% RSLogix 500 project TANK_ANAL_BAK001.RSS, saved by version 8.30.00.16 %
PROJECT "UNTITLED"    % processor: Bul.1763 MicroLogix 1100 Series B %

PROGRAM FILES
  LAD 2 "MAIN"  3 rungs
  LAD 3 "ANALOG IO"  4 rungs
  LAD 4 "CONTROLS"  5 rungs

DATA FILES
  O0 OUTPUT  5 elements
  I1 INPUT  14 elements
  S2 STATUS  66 elements
  B3 BINARY  1 elements
  T4 TIMER  2 elements
  C5 COUNTER  1 elements
  R6 CONTROL  1 elements
  N7 INTEGER  1 elements
  F8 FLOAT  1 elements

LADDER 2 "MAIN"
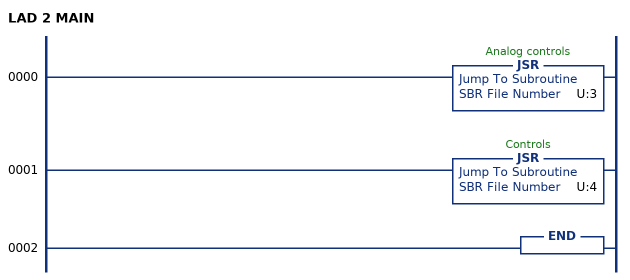
% Rung: 0 %
SOR JSR U:3 EOR
%   U:3  "Analog controls" %
% Rung: 1 %
SOR JSR U:4 EOR
%   U:4  "Controls" %
% Rung: 2 %
SOR END EOR

LADDER 3 "ANALOG IO"
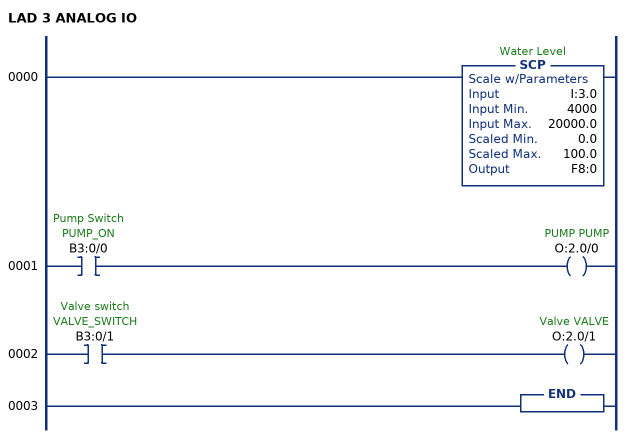
% Rung: 0 %
SOR SCP I:3.0 4000 20000.0 0.0 100.0 F8:0 EOR
%   I:3.0  WATER_LEVEL  "Water Level" %
%   F8:0  "Water Level" %
% Rung: 1 %
SOR XIC B3:0/0 OTE O:2.0/0 EOR
%   B3:0/0  PUMP_ON  "Pump Switch" %
%   O:2.0/0  PUMP  "PUMP" %
% Rung: 2 %
SOR XIC B3:0/1 OTE O:2.0/1 EOR
%   B3:0/1  VALVE_SWITCH  "Valve switch" %
%   O:2.0/1  VALVE  "Valve" %
% Rung: 3 %
SOR END EOR

LADDER 4 "CONTROLS"
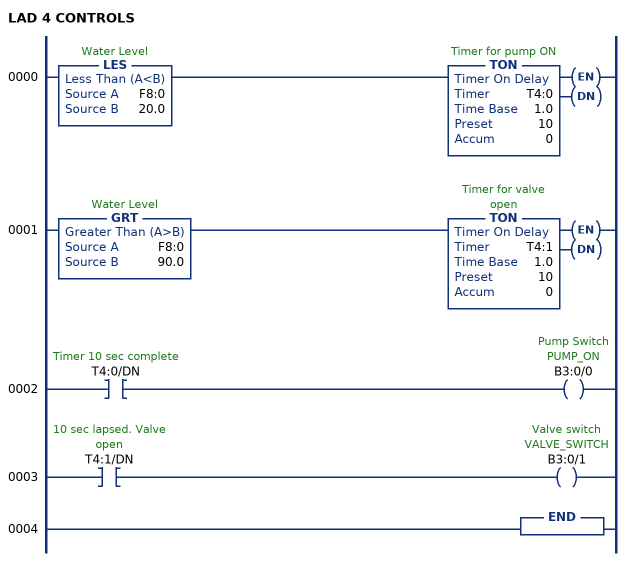
% Rung: 0 %
SOR LES F8:0 20.0 TON T4:0 1.0 10 0 EOR
%   F8:0  "Water Level" %
%   T4:0  "Timer for pump ON" %
% Rung: 1 %
SOR GRT F8:0 90.0 TON T4:1 1.0 10 0 EOR
%   F8:0  "Water Level" %
%   T4:1  "Timer for valve open" %
% Rung: 2 %
SOR XIC T4:0/DN OTE B3:0/0 EOR
%   T4:0/DN  "Timer 10 sec complete" %
%   B3:0/0  PUMP_ON  "Pump Switch" %
% Rung: 3 %
SOR XIC T4:1/DN OTE B3:0/1 EOR
%   T4:1/DN  "10 sec lapsed. Valve open" %
%   B3:0/1  VALVE_SWITCH  "Valve switch" %
% Rung: 4 %
SOR END EOR

OTHER DOCUMENTED ADDRESSES
  O:2.0  "WATER LEVEL OUT"

REVISION NOTES
  0: download

DATA TABLE (non-zero values as saved)
DATA T4
% .PRE .ACC %
% T4:0 % 10 0
% T4:1 % 10 0
